// TIA Portal V19 export
DATA_BLOCK "CallUnit_DB"   // DB54
// stored: InstanceOfName Unit2.CallUnit, InstanceOfType FB, Namespace Unit2
"Unit2.CallUnit"
   // VAR_INPUT
   //    safetyReleased { ExternalWritable := 'False'} : Bool;
   // END_VAR
   // VAR_OUTPUT
   //    acknowledgeSafety { ExternalWritable := 'False'} : Bool;
   // END_VAR
   // VAR_IN_OUT
   //    globalStatus : "LAF_typeGeneralStatus";
   //    unitInterface : "LAF_typeUnitInterface";
   // END_VAR
   // VAR
   //    statRemoteInterface { ExternalWritable := 'False'} : "LUC_typeCommands";
   //    instManageBitAlarms { ExternalWritable := 'False'} : "LAF_ManageBitAlarms";
   //    instStatusCollector { ExternalWritable := 'False'} : "LUC_StatusCollector";
   //    instInterfaceManager { ExternalWritable := 'False'} : "LUC_InterfaceManager";
   //    instUnitModeStateManager { ExternalWritable := 'False'} : "LPMLV2022_UnitModeStateManager";
   //    instRemoteInterfaceOpcUa { ExternalWritable := 'False'} : "LUC_RemoteCtrl_OpcUa";
   //    instSignalStack { ExternalWritable := 'False'} : "LUC_SignalStack";
   //    instUnitModeStateTimes { ExternalWritable := 'False'} : "LPMLV2022_UnitModeStateTimes";
   //    instLPMLV2022_UnitModeChangeAllowed { ExternalWritable := 'False'} : "LPMLV2022_UnitModeChangeAllowed";
   // END_VAR
BEGIN
END_DATA_BLOCK
